(*$
	Returns the current <a href="#mode_enum"><i>mode</i></a> of the instance <b><i>this</i></b>.
$*)
FUNCTION jog_manager_get_mode: mode_enum
VAR_IN_OUT
    CONVERSION_this:	jog_manager;	(*$ Instance to which the method applies $*)
END_VAR

jog_manager_get_mode := descriptor_get_mode(CONVERSION_this.descriptor);

END_FUNCTION

(* stored: Version 1.1.0.1, ProductVersion 3.1.4022.12
   POU jog_manager_get_mode: Id {ed495956-b2cd-45d4-9264-9189ad88fe74}, SpecialFunc None *)
